// LS Electric XG5000 project: 동남110
// PLC NewPLC
// module base 0 slot 0: 입출력 모듈:XBC-DN/DP14E (DC 24V 입력 8점, 트랜지스터 출력 6점)

PROGRAM NewProgram (task: 스캔 프로그램)

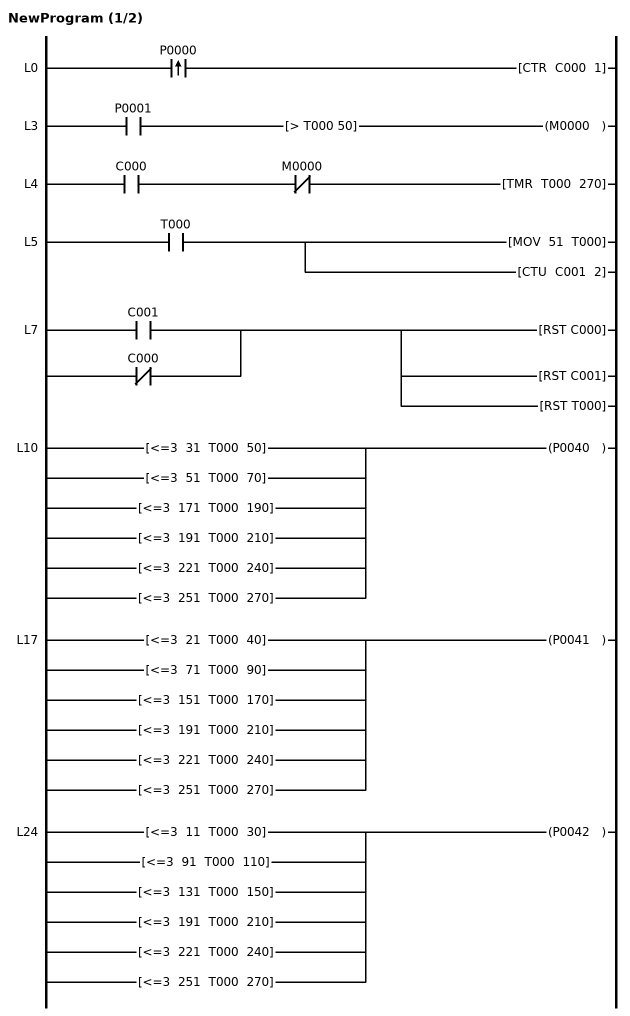
; L0
LOADP     P0000
CTR       C000 1
; L3
LOAD      P0001
AND>      T000 50
OUT       M0000
; L4
LOAD      C000
AND NOT   M0000
TMR       T000 270
; L5
LOAD      T000
MOV       51 T000
CTU       C001 2
; L7
LOAD      C001
OR NOT    C000
RST       C000
RST       C001
RST       T000
; L10
LOAD<=3   31 T000 50
OR<=3     51 T000 70
OR<=3     171 T000 190
OR<=3     191 T000 210
OR<=3     221 T000 240
OR<=3     251 T000 270
OUT       P0040
; L17
LOAD<=3   21 T000 40
OR<=3     71 T000 90
OR<=3     151 T000 170
OR<=3     191 T000 210
OR<=3     221 T000 240
OR<=3     251 T000 270
OUT       P0041
; L24
LOAD<=3   11 T000 30
OR<=3     91 T000 110
OR<=3     131 T000 150
OR<=3     191 T000 210
OR<=3     221 T000 240
OR<=3     251 T000 270
OUT       P0042

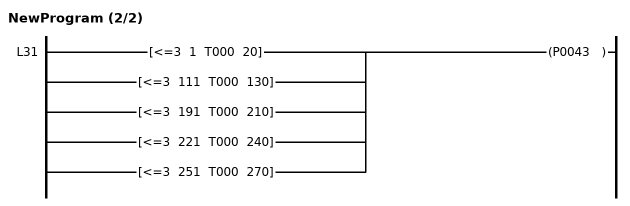
; L31
LOAD<=3   1 T000 20
OR<=3     111 T000 130
OR<=3     191 T000 210
OR<=3     221 T000 240
OR<=3     251 T000 270
OUT       P0043